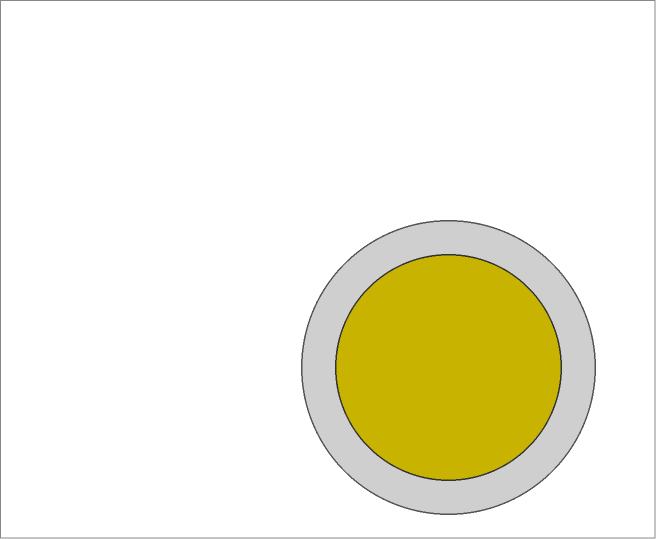
VISUALIZATION Visualization  // 656x539
    Lamp1 (241,196 415x343), variable: MAIN.bLed, style: Lamp-Lamp1-Yellow
END_VISUALIZATION

(* stored: Version 1.1.0.1
   Visu Visualization: Id {b7c72ae0-bcaa-4e87-9ead-939b5dcbd0f0} *)
